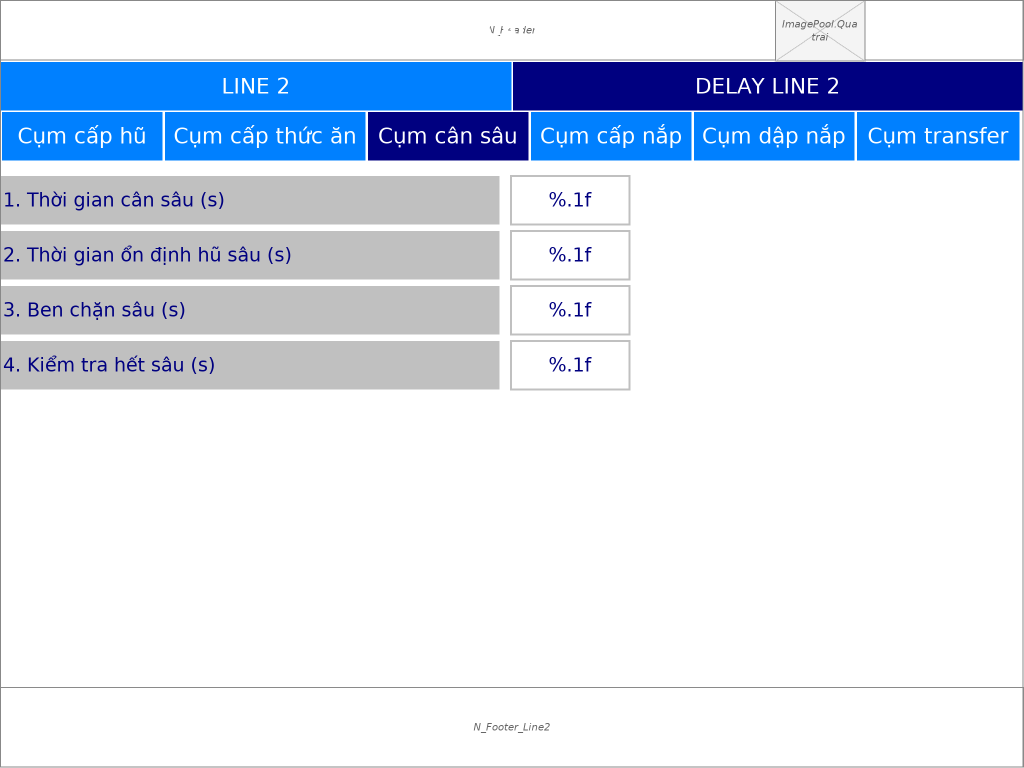
VISUALIZATION N_Setting_Delay_WorwWeight2  // 1024x768
    Frame (0,687 1024x80)
        shows N_Footer_Line2()
    Frame (0,0 1024x60)
        shows N_Header()
    Textfield (353,4 420x50), "MÀN HÌNH CÀI KHOẢNG TRỄ LINE 2"
    Rectangle (0,175 500x50), "1. Thời gian cân sâu (s)"
    Rectangle (0,285 500x50), "3. Ben chặn sâu (s)"
    Rectangle (0,230 500x50), "2. Thời gian ổn định hũ sâu (s)"
    Rectangle (0,61 512x50), "LINE 2"
        OnMouseClick: change screen: N_Setting_Line2
    Rectangle (1,111 162x50), "Cụm cấp hũ"
        OnMouseClick: change screen: N_Setting_Delay_JarSupply2
    Rectangle (164,111 202x50), "Cụm cấp thức ăn"
        OnMouseClick: change screen: N_Setting_Delay_FoodSupply2
    Rectangle (367,111 162x50), "Cụm cân sâu"
        OnMouseClick: change screen: N_Setting_Delay_WorwWeight2
    Rectangle (530,111 162x50), "Cụm cấp nắp"
        OnMouseClick: change screen: N_Setting_Delay_LidSupply2
    Rectangle (693,111 162x50), "Cụm dập nắp"
        OnMouseClick: change screen: N_Setting_Delay_LidPressing2
    Rectangle (856,111 164x50), "Cụm transfer"
        OnMouseClick: change screen: N_Setting_Delay_Tranfer2
    Rectangle (512,61 511x50), "DELAY LINE 2"
        OnMouseClick: change screen: N_Setting_Delay_JarSupply2
    Image (775,0 90x61), image: ImagePool.Qua trai
        OnMouseClick: change screen: N_Setting_Delay_WormWeight1
    Rectangle (510,285 120x50), "%.1f", text variable: PR_Line02.fTimer_Check_Cylinder
        OnMouseClick: write PR_Line02.fTimer_Check_Cylinder via VisuDialogs.Numpad
    Rectangle (510,230 120x50), "%.1f", text variable: PR_Line02.fTimer_Worm
        OnMouseClick: write PR_Line02.fTimer_Worm via VisuDialogs.Numpad
    Rectangle (510,175 120x50), "%.1f", text variable: PR_Line02.fTimer_Alarm_Worm
        OnMouseClick: write PR_Line02.fTimer_Alarm_Worm via VisuDialogs.Numpad
    Rectangle (0,340 500x50), "4. Kiểm tra hết sâu (s)"
    Rectangle (510,340 120x50), "%.1f", text variable: PR_Line02.fTimer_Error_Worm
        OnMouseClick: write PR_Line02.fTimer_Error_Worm via VisuDialogs.Numpad
END_VISUALIZATION

(* stored: Version 1.1.0.1, ProductVersion 3.1.4024.12
   Visu N_Setting_Delay_WorwWeight2: Id {c5eaaad4-921d-44fd-b30c-45704d1da764} *)
